Staubli VAL3: cycle.dtx

mdesc mNomSpeed
bool bIspower
public bool bIsEstop
num nWorkingStatus
num nWorkingMode
bool bConnected
public bool bCycle
public bool bPause
public bool bIsHome
public bool bRobotErr
public bool bIsRemote
public bool bConnected_Plc
string sIoBusStatus
num nJishu
num x_nResult
public bool bIsReady
string sMenu
num nPage
